FUNCTION_BLOCK EL4038
VAR
	_io : EL4xx8_Data;
	{attribute addProperty Name "WcState"}
	_wcState : WcStateBase;
	{attribute addProperty Name "Info data"}
	_infoData : InfoDataAds;
END_VAR

PROPERTY IO : REFERENCE TO EL4xx8_Data
GET
IO REF= _io;
END_GET
END_PROPERTY

PROPERTY WcState : REFERENCE TO WcStateBase
GET
WcState REF= _wcState;
END_GET
END_PROPERTY

END_FUNCTION_BLOCK

(* stored: Version 1.1.0.1, ProductVersion 3.1.4024.9
   POU EL4038: Id {ecd3e62d-af38-0ad8-1b86-7f8f568b499d}, SpecialFunc None
   Property IO: Id {e8e5d0ff-2b9f-0ba3-2102-34533d052965}
   Get Get: Id {1667cbdc-bc32-0ea9-2b86-62eba9b40f6d}
   Property WcState: Id {96dcc8cb-f9fe-054d-2bb6-9c87d3565b54}
   Get Get: Id {0cbca103-483b-0ac3-2fee-f0acb0ccabb6} *)
